(* IEC 61131-3 sources: horner-cscape-mcp/artifacts/projects/HashTestProj/pous, 1 file *)

(* ---- HashPOU.st ---- *)
PROGRAM HashTest
VAR
    y : INT;
END_VAR
y := 99;
END_PROGRAM
